{attribute addProperty BoxType "EL3403-0000-0018"}
{attribute addProperty Id "PM_Inputs_ChannelAT %I*ARRAY[0..14] OF PM_Inputs_Channel_2B79FE26456570PM_Status_dataAT %I*PM_Status_data_CC42570F4050PM_Outputs_ChannelAT %Q*ARRAY[0..2] OF PM_Outputs_Channel_A1108FBB2430WcStateAT %I*WcState_98A4DF7520.250InfoDataAT %I*InfoData_BC63D37F80100"}
{attribute addProperty CRC "464351516"}
{attribute addProperty SizeInBites "602"}
{attribute addProperty SizeInBytes "75.25"}
TYPE EL3403_602DA439 :
STRUCT
	{attribute addProperty Name "PM_Inputs_Channel"}
	PM_Inputs_Channel : ARRAY[0..14] OF PM_Inputs_Channel_2B79FE26;
	{attribute addProperty Name "PM_Status_data"}
	PM_Status_data : PM_Status_data_CC42570F;
	{attribute addProperty Name "PM_Outputs_Channel"}
	PM_Outputs_Channel : ARRAY[0..2] OF PM_Outputs_Channel_A1108FBB;
	{attribute addProperty Name "WcState"}
	WcState : WcState_98A4DF75;
	{attribute addProperty Name "InfoData"}
	InfoData : InfoData_BC63D37F;
END_STRUCT
END_TYPE

(* stored: Version 1.2.0.0, ProductVersion 3.1.4024.9
   DUT EL3403_602DA439: Id {a6e4a4f2-ea7c-4e1a-8076-853bf903d10f} *)
